# EPICS autosave request: iocBoot/iocUSB1808/auto_settings.req
file "USB1808_settings.req", P=$(P)
